Universal Robots PolyScope program: Rotation around Z.urp

ProgramRoot directory=/home/ur/ursim-3.1/programs/Support site; kinematics=(a=[0, -0.425, -0.39243, 0, 0, 0], d=[0.0892, 0, 0, 0.109, 0.093, 0.082], alpha=[1.5708, 0, 0, 1.5708, -1.5708, 0], deltaTheta=[0, 0, 0, 0, 0, 0], status=notInitialized); lastSavedInVersion=(project__name=Polyscope, major__version=3, minor__version=1, svn__revision=18024, build__date=Jul 07 2015, 15:18:49); name=Rotation around Z; programVersion=(project__name=PolyScope, major__version=1, minor__version=5, svn__revision=7849, build__date=Feb 06 2012, 15:16:46); robotEnvironmentFileName=default; serialNumberRobot=2015350001
  MainProgram cartesianAcceleration=1.2; cartesianSpeed=0.25; jointAcceleration=1.3962634015954636; jointSpeed=1.0471975511965976; sharedProcessMoveBlendRadius=0.025; motionType=JOINT_SPACE
    Move cartesianAcceleration=1.2; cartesianSpeed=0.25; jointAcceleration=1.3962634015954636; jointSpeed=1.0471975511965976; sharedProcessMoveBlendRadius=0.025; motionType=JOINT_SPACE
      Waypoint blendRadius=0.0; cartesianAcceleration=1.2; cartesianSpeed=0.25; jointAcceleration=1.3962634015954636; jointSpeed=1.0471975511965976; nextMotionTime=2.0; useSharedBlendParameter=true; useSharedParameters=true; outputFlangePose=(pos=(x=-0.3012933420675599, y=-0.3009734881857273, z=0.09982168694612403), rot=(x=-2.695833833015667, y=1.6053216080568666, z=-0.03655853624804491)); position=TCP in base x=-300.031 y=-300.068 z=100.037 mm, rx=-2.6958 ry=1.6053 rz=-0.0366 rad; joints [29.907, -77.52, 132.345, -143.983, 271.058, 181.446] deg; positionType=FIXED_POSITION; waypointPoseInFeatureCoordinates=(pos=(x=-0.3000311766275814, y=-0.30006806343793485, z=0.100036731612092), rot=(x=-2.6958266290097836, y=1.6053174771728282, z=-0.03656568316875425)); name=Waypoint_1
    Assignment expr=get_actual_tcp_pose(); operatorValueType=INTEGER; valueSource=EXPRESSION
    Assignment expr=d2r(90); operatorValueType=INTEGER; valueSource=EXPRESSION
    Assignment expr=pose_trans(ExpressionVariableNode,p[0,0,0,0,0,ExpressionVariableNode]); operatorValueType=INTEGER; valueSource=EXPRESSION
    Move cartesianAcceleration=1.2; cartesianSpeed=0.25; jointAcceleration=1.3962634015954636; jointSpeed=1.0471975511965976; sharedProcessMoveBlendRadius=0.025; motionType=CARTESIAN_SPACE
      Waypoint blendRadius=0.05; cartesianAcceleration=1.2; cartesianSpeed=0.25; jointAcceleration=1.3962634015954636; jointSpeed=1.0471975511965976; nextMotionTime=2.0; stoppoint=true; useSharedBlendParameter=true; useSharedParameters=true; positionType=VARIABLE_POSITION; name=Waypoint
      Popup message=Stop; type=MESSAGE
    Wait 
